(* Logix 5000 project; controller FRIST_EXAMPLE Emulate 5570 rev 19.11; software revision 19.01 *)

TASK MainTask (continuous, watchdog 500 ms) : MainProgram

MODULES
   Local : Emulate 5570 (ICP 2, rev 19.11)
       : 1756-IB32 (ICP 3, rev 3.1, Input RPI 20 ms)   // DG-INPUT
       : vendor 1 type 7 code 8 (ICP 4, rev 3.1, Output RPI 20 ms)
       : 1756-IF6I (ICP 5, rev 1.1, Input RPI 100 ms)
       : 1756-OF8 (ICP 6, rev 1.1, Output RPI 12 ms)
END_MODULES

VAR_GLOBAL   (* controller tags *)
   CMD_MT01 : BOOL;
   DESLIGA : BOOL := 1;
   LIGA : BOOL;
END_VAR

PROGRAM MainProgram   (* main routine MainRoutine *)
VAR
   aux1 : REAL := 25.0;
   BT_DESLIGA : BOOL;
   BT_LIGA : BOOL;
   HIGHT_LEVEL : BOOL;
   LIT01 : REAL;   // Valor Escalonado
   LOW_LEVEL : BOOL := 1;
   m : REAL := 0.00625;   // Coef. Ang. Reta
   MOTOR01 : BOOL := 1;
   SP_HIGHT : REAL := 80.0;   // Set Point Alto
   SP_LOW : REAL := 20.0;
END_VAR

ROUTINE MainRoutine   (* ladder *)
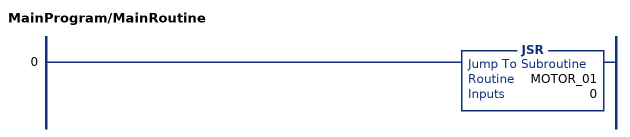
   0: JSR(MOTOR_01,0);
END_ROUTINE

ROUTINE MOTOR_01   (* ladder *)
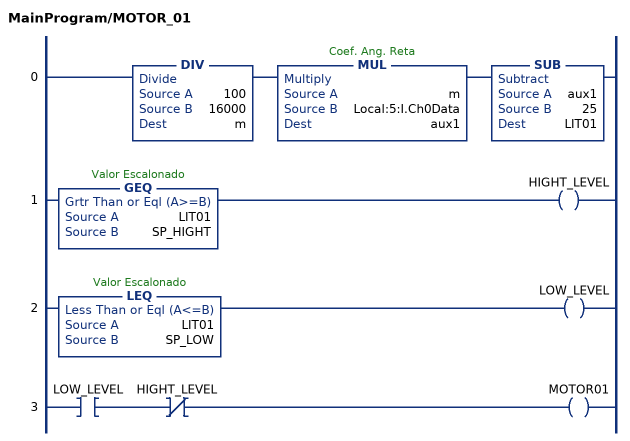
   0: DIV(100,16000,m)MUL(m,Local:5:I.Ch0Data,aux1)SUB(aux1,25,LIT01);
   1: GEQ(LIT01,SP_HIGHT)OTE(HIGHT_LEVEL);
   2: LEQ(LIT01,SP_LOW)OTE(LOW_LEVEL);
   3: XIC(LOW_LEVEL)XIO(HIGHT_LEVEL)OTE(MOTOR01);
END_ROUTINE
END_PROGRAM
